// TIA Portal project "Control Nivel de Tanque" (V17)

(* hardware
DEVICE "S7-1200 station_1"  S7-1200 Station
   slot 0: "Rack_0"  S7-1200 Rack  Rack  V1.0
   slot 1: "PLC_1"  CPU 1212C AC/DC/Rly  6ES7 212-1BE40-0XB0  V4.5
*)

// ===== PLC "PLC_1"  CPU 1212C AC/DC/Rly =====

VAR_GLOBAL   // PLC tag table "Perifericos"
   "Start" AT %I3.0 : Bool;
   "Stop" AT %I3.1 : Bool;
   "ParoEmergencia" AT %I3.2 : Bool;
   "LT1" AT %I3.3 : Bool;
   "LT2" AT %I3.4 : Bool;
   "LT3" AT %I3.5 : Bool;
   "V1" AT %Q4.0 : Bool;
   "V2" AT %Q4.1 : Bool;
   "Motor" AT %Q4.2 : Bool;
   "Encendido" AT %M10.0 : Bool;
END_VAR

FUNCTION "MHJ-PLC-Lab-Function-S71200" : Void   // FC9000, SCL
{ S7_Optimized_Access := 'TRUE' }
VERSION : 0.1
   VAR_TEMP
      rdTimeReturn : Int;
      outputTime : DTL;
      SyncVal : Byte;
      forVal : Int;
      forVal_2 : Int;
      Value : Byte;
   END_VAR
   VAR CONSTANT
      CompVal : Byte := 16#34;
      Value_01 : Byte := 16#11;
      Value_01_DW : DWord := 16#A165_D992;
      Value_02_DW : DWord := 16#58BE_4401;
   END_VAR
BEGIN

   #Value:=PEEK(area := 16#82,
        dbNumber := 0,
        byteOffset := 511);
   #Value := #Value + 1;

   POKE(area := 16#82,
        dbNumber := 0,
        byteOffset := 511,
        value := #Value);

   POKE(area:=16#81,
        dbNumber:=0,
        byteOffset:=1016,
        value:=#Value_01_DW);
   POKE(area := 16#81,
        dbNumber := 0,
        byteOffset := 1020,
        value := #Value_02_DW);

   POKE(area := 16#81,
        dbNumber := 0,
        byteOffset := 511,
        value := B#16#00);

   FOR #forVal := 0 TO 120 DO
       FOR #forVal_2:=0 TO 10 DO
           #rdTimeReturn:=RD_SYS_T(#outputTime);
           #rdTimeReturn := WR_SYS_T(#outputTime);
           #rdTimeReturn := RD_SYS_T(#outputTime);
           #rdTimeReturn := WR_SYS_T(#outputTime);
       END_FOR;
       #SyncVal:= PEEK(area := 16#81,
                      dbNumber := 0,
                      byteOffset := 511);
       IF #SyncVal = #CompVal THEN
          GOTO M_1;
       END_IF;
   END_FOR;
   RETURN;

   M_1:
   POKE(area := 16#81,
        dbNumber := 0,
        byteOffset := 511,
        value := B#16#0);
END_FUNCTION

ORGANIZATION_BLOCK "Main"   // OB1, LAD, ProgramCycle
TITLE = "Main Program Sweep (Cycle)"
{ S7_Optimized_Access := 'TRUE' }
VERSION : 0.1
   VAR_INPUT
      Initial_Call : Bool;   // Initial call of this OB
      Remanence : Bool;   // =True, if remanent data are available
   END_VAR
BEGIN

REGION Network 1
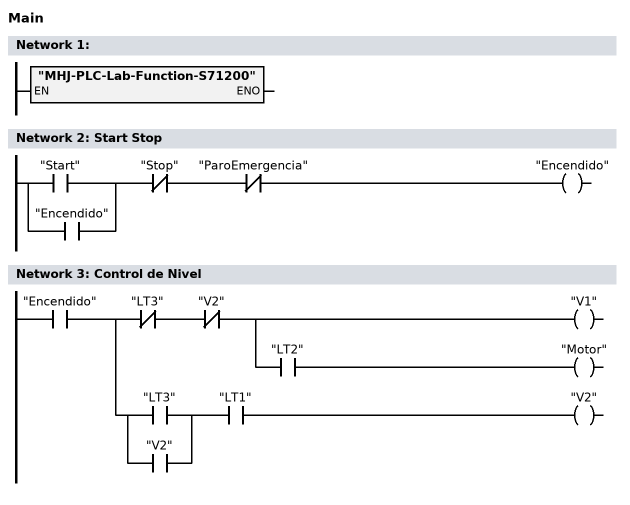
   RUNG wire#powerrail
      "MHJ-PLC-Lab-Function-S71200"()
   END_RUNG
   // the same network as SCL:
   "MHJ-PLC-Lab-Function-S71200"();
END_REGION

REGION Network 2: Start Stop
   RUNG wire#powerrail
      Contact( "Start" )
      wire#w1
      I_Contact( "Stop" )
      I_Contact( "ParoEmergencia" )
      Coil( "Encendido" )
   END_RUNG
   RUNG wire#powerrail
      Contact( "Encendido" )
   END_RUNG wire#w1
   // the same network as SCL:
   "Encendido" := ("Start" OR "Encendido") AND NOT "Stop" AND NOT "ParoEmergencia";
END_REGION

REGION Network 3: Control de Nivel
   RUNG wire#powerrail
      Contact( "Encendido" )
      wire#w1
      I_Contact( "LT3" )
      I_Contact( "V2" )
      wire#w2
      Coil( "V1" )
   END_RUNG
   RUNG wire#w2
      Contact( "LT2" )
      Coil( "Motor" )
   END_RUNG
   RUNG wire#w1
      Contact( "LT3" )
      wire#w3
      Contact( "LT1" )
      Coil( "V2" )
   END_RUNG
   RUNG wire#w1
      Contact( "V2" )
   END_RUNG wire#w3
   // the same network as SCL:
   "V1" := "Encendido" AND NOT "LT3" AND NOT "V2";
   "Motor" := "V1" AND "LT2";
   "V2" := "Encendido" AND ("LT3" OR "V2") AND "LT1";
END_REGION
END_ORGANIZATION_BLOCK